// Mitsubishi GX Works2 project: 2015.03.20voice   PLC: FX1N/FX1NC

PROGRAM MAIN
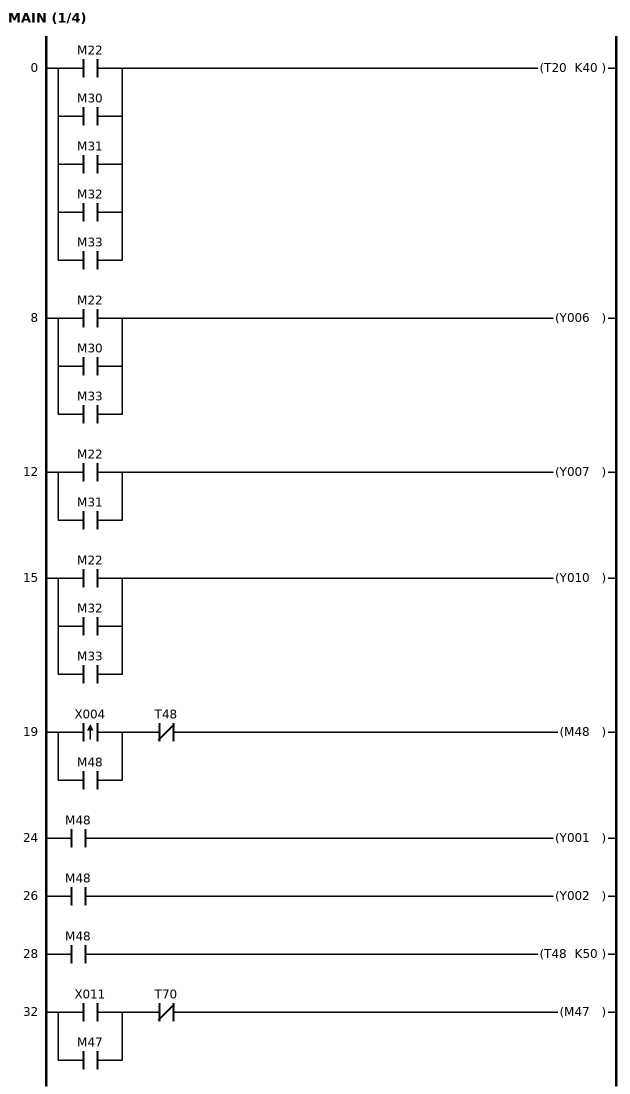
0     LD      M22
      OR      M30
      OR      M31
      OR      M32
      OR      M33
      OUT     T20 K40
8     LD      M22
      OR      M30
      OR      M33
      OUT     Y006
12    LD      M22
      OR      M31
      OUT     Y007
15    LD      M22
      OR      M32
      OR      M33
      OUT     Y010
19    LDP     X004
      OR      M48
      ANI     T48
      OUT     M48
24    LD      M48
      OUT     Y001
26    LD      M48
      OUT     Y002
28    LD      M48
      OUT     T48 K50
32    LD      X011
      OR      M47
      ANI     T70
      OUT     M47
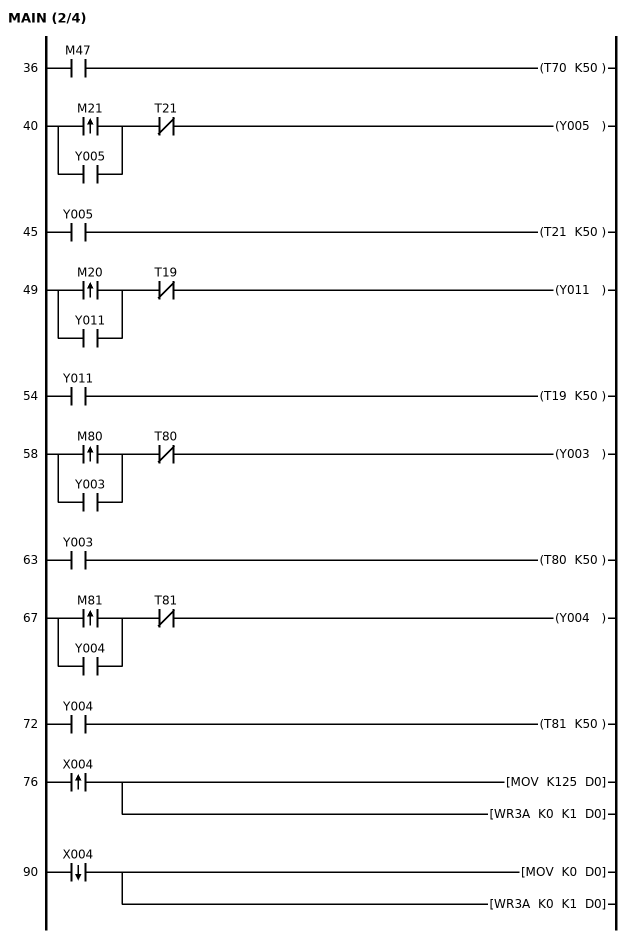
36    LD      M47
      OUT     T70 K50
40    LDP     M21
      OR      Y005
      ANI     T21
      OUT     Y005
45    LD      Y005
      OUT     T21 K50
49    LDP     M20
      OR      Y011
      ANI     T19
      OUT     Y011
54    LD      Y011
      OUT     T19 K50
58    LDP     M80
      OR      Y003
      ANI     T80
      OUT     Y003
63    LD      Y003
      OUT     T80 K50
67    LDP     M81
      OR      Y004
      ANI     T81
      OUT     Y004
72    LD      Y004
      OUT     T81 K50
76    LDP     X004
      MOV     K125 D0
      WR3A    K0 K1 D0
90    LDF     X004
      MOV     K0 D0
      WR3A    K0 K1 D0
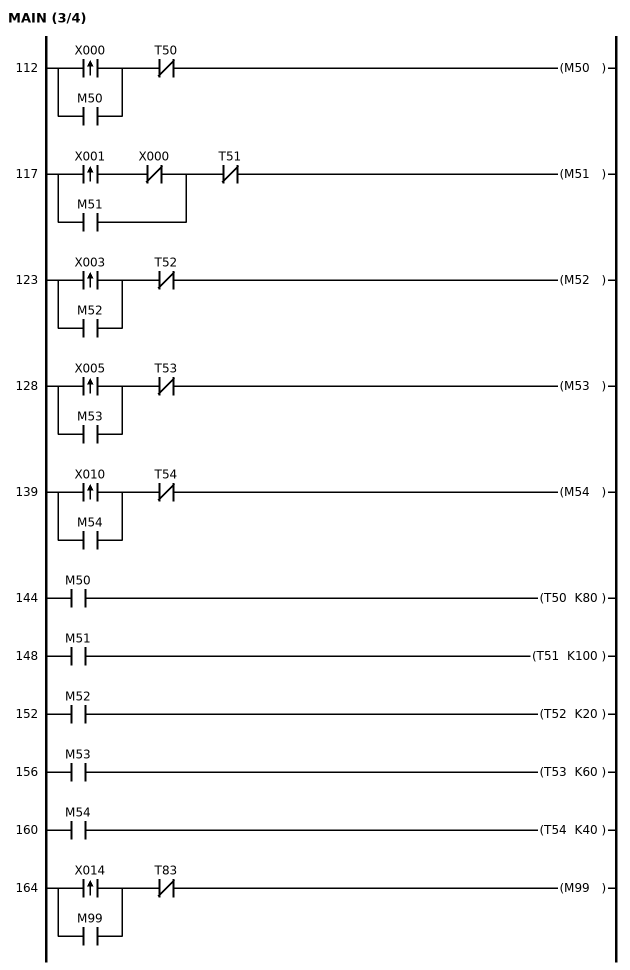
112   LDP     X000
      OR      M50
      ANI     T50
      OUT     M50
117   LDP     X001
      ANI     X000
      OR      M51
      ANI     T51
      OUT     M51
123   LDP     X003
      OR      M52
      ANI     T52
      OUT     M52
128   LDP     X005
      OR      M53
      ANI     T53
      OUT     M53
139   LDP     X010
      OR      M54
      ANI     T54
      OUT     M54
144   LD      M50
      OUT     T50 K80
148   LD      M51
      OUT     T51 K100
152   LD      M52
      OUT     T52 K20
156   LD      M53
      OUT     T53 K60
160   LD      M54
      OUT     T54 K40
164   LDP     X014
      OR      M99
      ANI     T83
      OUT     M99
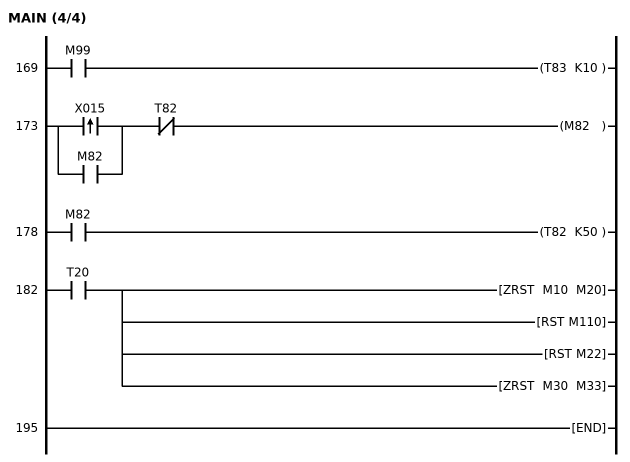
169   LD      M99
      OUT     T83 K10
173   LDP     X015
      OR      M82
      ANI     T82
      OUT     M82
178   LD      M82
      OUT     T82 K50
182   LD      T20
      ZRST    M10 M20
      RST     M110
      RST     M22
      ZRST    M30 M33
195   END
END_PROGRAM
